Fanuc KAREL source: kf00029.KL

-- PROVISIONAL review KL for V770-1; original PC SHA256 911f201a4a50c263f4d3f84d1a65943da835775ece831ee5824aa59f51ca7bf8
-- Incomplete behavior may be omitted. Consult companion uncertainty JSON. Do not deploy.
PROGRAM KF00029
%NOLOCKGROUP
VAR
  I : INTEGER
  J : INTEGER
  X : REAL
  Y : REAL
  B : BOOLEAN
  C : BOOLEAN
  TXT : STRING[80]
  TXT2 : STRING[80]
  STATUS : INTEGER
-- UNRESOLVED_DECL AI type=002010
-- UNRESOLVED_DECL BI type=002010
-- UNRESOLVED_DECL P type=000102
-- UNRESOLVED_DECL JP type=000199
-- UNRESOLVED_DECL PF type=000101
-- UNRESOLVED_DECL V1 type=000013
-- UNRESOLVED_DECL V2 type=000013
BEGIN
  -- UNRESOLVED_PC offsets 5-12; opcodes 9D,23
  -- UNRESOLVED_PC offsets 17-24; opcodes 9C,23
  -- UNRESOLVED_PC offsets 29-48; opcodes 21,21,47,23
  -- UNRESOLVED_PC offsets 53-57; opcodes 7F
END KF00029
